// TIA Portal V19 export
DATA_BLOCK "INTERLOCK DB"   // DB4
{ S7_Optimized_Access := 'TRUE' }
// stored: MemoryReserve 100
BEGIN
END_DATA_BLOCK
